(*

.. <legal notes>

legal notes
=================
| SPDX-FileCopyrightText: © 2026 Oleksandr Tiutyk <trofimich@gmail.com>
| SPDX-License-Identifier: LGPL-3.0-only
| For details check: LGPL-3.0-only_

.. _LGPL-3.0-only: https://www.gnu.org/licenses/lgpl-3.0.en.html

.. </legal notes>

*)

INTERFACE IDynamicDictionary EXTENDS IReadOnlyDynamicDictionary

METHOD Clear : IDynamicDictionary
END_METHOD

METHOD RemoveAt : IDynamicDictionary
VAR_INPUT
	index : DINT;
END_VAR
END_METHOD

METHOD SetCopy : IDynamicDictionary
VAR_INPUT
	key : ANY;
	value : ANY;
	keyIsObject : BOOL := FALSE;
	valueIsObject : BOOL := FALSE;
END_VAR
VAR_OUTPUT
	index : DINT;
END_VAR
END_METHOD

METHOD SetGeneric : IDynamicDictionary
VAR_INPUT
	key : GENERIC_VALUE;
	value : GENERIC_VALUE;
END_VAR
VAR_OUTPUT
	index : DINT;
END_VAR
END_METHOD

METHOD TryRemoveByGenericKey : IDynamicDictionary
VAR_INPUT
	key : GENERIC_VALUE;
	releaseKey : BOOL := TRUE;
END_VAR
VAR_OUTPUT
	removed : BOOL;
END_VAR
END_METHOD

METHOD TryRemoveByKey : IDynamicDictionary
VAR_INPUT
	key : ANY;
END_VAR
VAR_OUTPUT
	removed : BOOL;
END_VAR
END_METHOD

END_INTERFACE

(* stored: Version 1.1.0.1
   Itf IDynamicDictionary: Id {57e81792-3900-4cad-861e-9c1a745a287a}
   Method Clear: Id {b1563b71-bd6a-4263-830c-984583112e42}
   Method RemoveAt: Id {a1586ec5-b74e-4671-96ad-ae4197067882}
   Method SetCopy: Id {f13fbbaa-2923-411c-9a7c-638998bcf36d}
   Method SetGeneric: Id {9a515aa5-db44-4d5d-9fbd-7695318ffa56}
   Method TryRemoveByGenericKey: Id {ed98c14c-8b20-4e0c-b155-925d2858a0a4}
   Method TryRemoveByKey: Id {2539d3ce-1d3f-4331-818e-1181097b6910} *)
